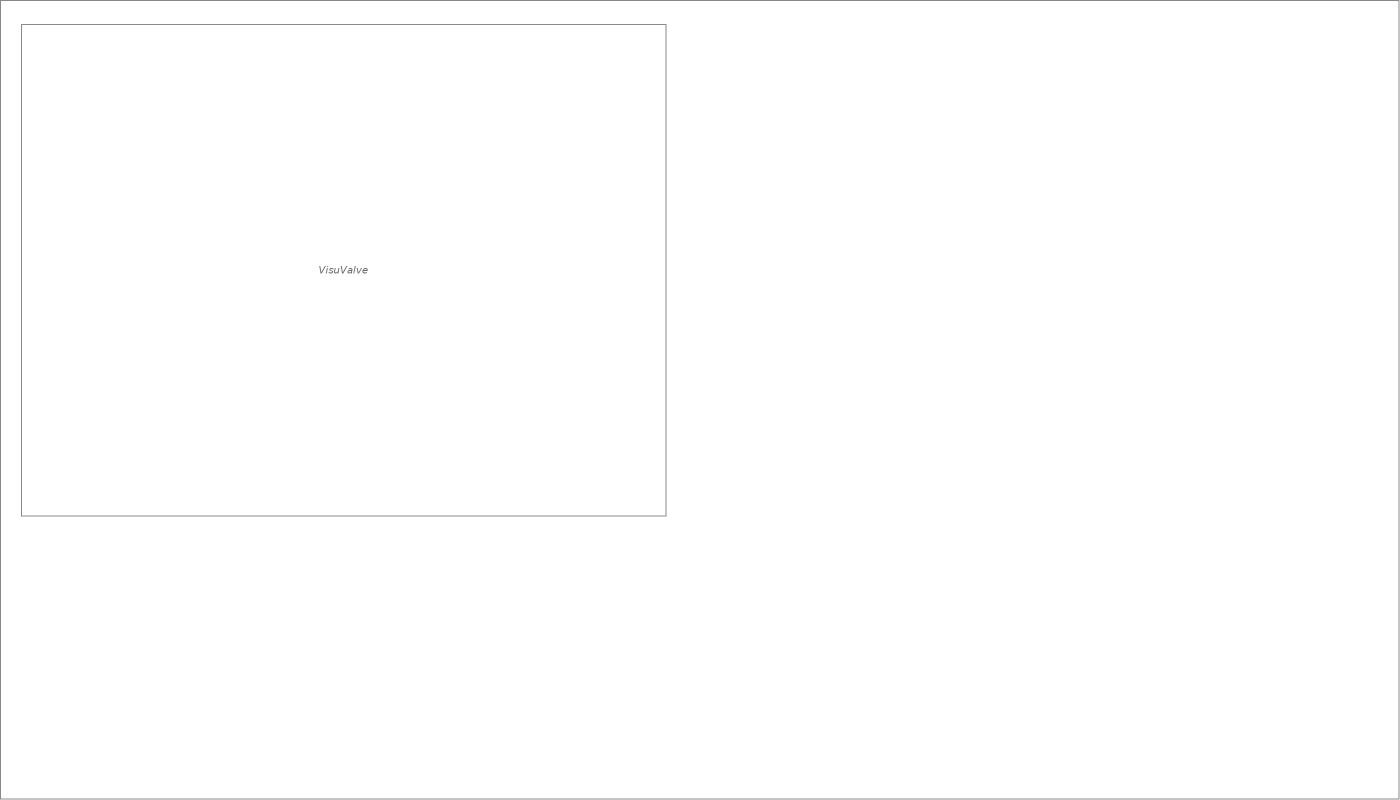
VISUALIZATION VisuMain  // 1400x800
    Frame (21,24 645x492)
        shows VisuValve()
        p2584409864: GVL_VCM.valve01
        p1828834575: GVL_VCM.ioValve01
END_VISUALIZATION

(* stored: Version 1.1.0.1, ProductVersion 3.1.4024.12
   Visu VisuMain: Id {459736cf-f2d9-4d2f-916e-a2ee046ee317} *)
